PROGRAM SelectSpike
VAR
	current_pos: ARRAY [1..5] OF WORD :=[16#4355, 16#5252, 16#454E, 16#5420, 16#504F];
	pos: ARRAY [1..5] OF WORD := [16#5320, 16#2020, 16#2020, 16#2020, 16#2020];

	row: ARRAY [1..10] OF WORD;
	indexs: ARRAY [1..GV_HMI.iMaxTargets] OF INT;
	found: BOOL := FALSE;
	
	indexesIndex: INT := 1;
	firstSpikeIndex: INT := 0;
	secondSpikeIndex: INT := 0;
	thirdSpikeIndex: INT := 0;	
	
	selectedCursorIndex: INT := 0;	
	cursorIndex: INT := 1;
	lastPos : REAL := GV_LIFT.TARGET_POSITION;
	noneSelectedTargetPosValue : REAL := 0;
	
END_VAR

IF GV_MODBUS.btnData = GV_MODBUS.btnUp THEN
	cursorIndex:= cursorIndex - 1;
	selectedCursorIndex := 0;
	GV_HMI.TargetPos := noneSelectedTargetPosValue;
	Execute_Write_Screen();
END_IF

IF GV_MODBUS.btnData = GV_MODBUS.btnDwn THEN
	cursorIndex:= cursorIndex + 1;	
	selectedCursorIndex := 0;
	GV_HMI.TargetPos := noneSelectedTargetPosValue;
	Execute_Write_Screen();	
END_IF

IF NOT GV_MODBUS.wasMTS THEN
	selectedCursorIndex := 0;
	GV_HMI.TargetPos := noneSelectedTargetPosValue;
END_IF

IF GV_MODBUS.btnData = GV_MODBUS.btnEnter THEN
	selectedCursorIndex := cursorIndex;
	
	IF cursorIndex = 1 THEN
		GV_LIFT.TARGET_POSITION := XML.savedvalues.savedpos[firstSpikeIndex].target;
	ELSIF cursorIndex = 2 THEN
		GV_LIFT.TARGET_POSITION := XML.savedvalues.savedpos[secondSpikeIndex].target;
	ELSIF cursorIndex = 3 THEN
		GV_LIFT.TARGET_POSITION := XML.savedvalues.savedpos[thirdSpikeIndex].target;
	END_IF
	
	Execute_Write_Screen();
END_IF

indexs := Get_Valid_Indexs();

IF firstSpikeIndex = 0 THEN
	firstSpikeIndex := indexs[1];
	secondSpikeIndex := indexs[2];
	thirdSpikeIndex := indexs[3];
END_IF

IF cursorIndex < 1 THEN
	indexesIndex := indexesIndex - 1;
	
	IF indexesIndex < 1 THEN
		indexesIndex := 1;
	END_IF
	
	firstSpikeIndex := indexs[indexesIndex];
	secondSpikeIndex := indexs[indexesIndex + 1];
	thirdSpikeIndex := indexs[indexesIndex + 2];
	
	cursorIndex := 1;
END_IF

IF cursorIndex > 3 THEN	
	indexesIndex := indexesIndex + 1;
	
	IF indexesIndex > (GV_HMI.iMaxTargets - 2) THEN
		indexesIndex := GV_HMI.iMaxTargets - 2;
	END_IF
	
	IF indexs[indexesIndex + 2] = 0 THEN
		indexesIndex := indexesIndex - 1;
	END_IF
	
	IF indexesIndex < 1 THEN
		indexesIndex := 1;
	END_IF
		
	firstSpikeIndex := indexs[indexesIndex];
	secondSpikeIndex := indexs[indexesIndex + 1];
	thirdSpikeIndex := indexs[indexesIndex + 2];
	
	cursorIndex := 3;
END_IF

GV_MODBUS.oneLeft:= current_pos;         
GV_MODBUS.oneRight:= GV_MODBUS.blank;
GV_MODBUS.twoLeft:= GV_MODBUS.blank;
GV_MODBUS.twoRight:= GV_MODBUS.blank;
GV_MODBUS.threeLeft:= GV_MODBUS.blank;
GV_MODBUS.threeRight:= GV_MODBUS.blank;	
GV_MODBUS.fourLeft:= GV_MODBUS.blank; 
GV_MODBUS.fourRight:= GV_MODBUS.blank;

GV_MODBUS.oneRight:= Position_To_Row_Array(pos, GV_LIFT.CURRENT_POSITION);     
	
IF firstSpikeIndex > 0 THEN		
	IF XML.savedvalues.savedpos[firstSpikeIndex].target < GV_MODBUS.filterTarget THEN
		
		
		IF cursorIndex = 1 AND NOT (selectedCursorIndex = 1) THEN
			row := Spike_To_Row_Array(GV_MODBUS.selectedASCII, XML.savedvalues.savedpos[firstSpikeIndex]);
		ELSIF selectedCursorIndex = 1 THEN
			row := Spike_To_Row_Array(GV_MODBUS.loadedASCII, XML.savedvalues.savedpos[firstSpikeIndex]);
		ELSE
			row := Spike_To_Row_Array(GV_MODBUS.spaceASCII, XML.savedvalues.savedpos[firstSpikeIndex]);
		END_IF
		
		Fill_Row_Two(row);
	END_IF
END_IF
	
IF secondSpikeIndex > 0 THEN					   
	IF XML.savedvalues.savedpos[secondSpikeIndex].target < GV_MODBUS.filterTarget THEN
		
		
		IF cursorIndex = 2 AND NOT (selectedCursorIndex = 2) THEN
			row := Spike_To_Row_Array(GV_MODBUS.selectedASCII, XML.savedvalues.savedpos[secondSpikeIndex]);		
		ELSIF selectedCursorIndex = 2 THEN
			row := Spike_To_Row_Array(GV_MODBUS.loadedASCII, XML.savedvalues.savedpos[secondSpikeIndex]);	
		ELSE
			row := Spike_To_Row_Array(GV_MODBUS.spaceASCII, XML.savedvalues.savedpos[secondSpikeIndex]);
		END_IF
		 
		Fill_Row_Three(row);
	END_IF	
END_IF

IF thirdSpikeIndex > 0 THEN
	IF XML.savedvalues.savedpos[thirdSpikeIndex].target < GV_MODBUS.filterTarget THEN
		IF cursorIndex = 3 AND NOT (selectedCursorIndex = 3) THEN
			row := Spike_To_Row_Array(GV_MODBUS.selectedASCII, XML.savedvalues.savedpos[thirdSpikeIndex]); 				
		ELSIF selectedCursorIndex = 3 THEN
			row := Spike_To_Row_Array(GV_MODBUS.loadedASCII, XML.savedvalues.savedpos[thirdSpikeIndex]);
		ELSE
			row := Spike_To_Row_Array(GV_MODBUS.spaceASCII, XML.savedvalues.savedpos[thirdSpikeIndex]); 
		END_IF
		
		Fill_Row_Four(row);				
	END_IF
END_IF

IF NOT GV_MODBUS.readExecute AND GV_MODBUS.addr = GV_MODBUS.oneLeftAddr THEN
	GV_MODBUS.data:= GV_MODBUS.oneLeft;
END_IF

END_PROGRAM

(* stored: Version 1.1.0.1, ProductVersion 3.1.4022.12
   POU SelectSpike: Id {3400e5d8-f531-4690-b110-580b0ceb5e1c}, SpecialFunc None *)
